FUNCTION_BLOCK FB_Stopcontact
VAR
	Output			: Stopcontact_output;
	kWh_meter		: FB_Verbruikmeter;
	
END_VAR

END_FUNCTION_BLOCK

(* stored: Version 1.1.0.1, ProductVersion 3.1.4024.12
   POU FB_Stopcontact: Id {4f4e8c13-b316-4d55-9d9a-01d11f7ddfdd}, SpecialFunc None *)
